TEXTLIST Energy_Meters_Status
  0 = 'Ok'
  1 = 'Error'
  2 = 'Alarm'
   = ''
END_TEXTLIST

(* stored: Version 1.1.0.1, ProductVersion 3.1.4024.12
   TextList Energy_Meters_Status: Id {c03bfe82-9829-4fa0-b4ac-e1f2820692d0} *)
